TYPE ST_HMIWebDriveStatus EXTENDS ST_HMIStatus :
STRUCT
	DriveState : Motion.E_WebDriveState;
	Calibrated : BOOL;
	TensionerRadius : LREAL;
	TensionerTension : LREAL;
	WinderRadius : LREAL;
END_STRUCT
END_TYPE

(* stored: Version 1.1.0.1
   DUT ST_HMIWebDriveStatus: Id {7c628b72-9457-4b4b-b959-b4a70f39a9bf} *)
